(* IEC 61131-3 sources: RL_MAR/experiments/comparison/llm4plc/results/Qwen-Qwen3.5-9B_20260506_150728/20260506_170933, 3 files *)

(* ---- generated_code_iteration_0.st ---- *)
START_ST
FUNCTION_BLOCK BakeryOvenControl
VAR_INPUT
    TemperatureSensor : REAL; (* Sensor input for oven temperature *)
    HumiditySensor : REAL; (* Sensor input for oven humidity *)
    StartSignal : BOOL; (* Input to start the baking process *)
END_VAR
VAR_OUTPUT
    HeatingElement : BOOL; (* Control signal for heating element *)
    CoolingElement : BOOL; (* Control signal for cooling element *)
    HumidityControl : BOOL; (* Control signal for humidity system *)
    DehumidityControl : BOOL; (* Control signal for dehumidification *)
END_VAR
VAR
    OvenTemperature : REAL := 0.0; (* Current oven temperature setpoint *)
    OvenHumidity : REAL := 0.0; (* Current humidity setpoint *)
    BakingTime : TIME := T#0s; (* Total baking time setpoint *)
    OvenStatus : BOOL := FALSE; (* Oven status: TRUE=On, FALSE=Off *)
    HeatingThreshold : REAL := 2.0; (* Temperature control threshold *)
    HumidityThreshold : REAL := 5.0; (* Humidity control threshold *)

    CurrentTemperature : REAL; (* To store the latest sensor reading *)
    CurrentHumidity : REAL; (* To store the latest sensor reading *)
    TimerAccumulator : TIME := T#0s; (* To accumulate time for the 1-second decrement logic *)
    TimerFlag : BOOL := FALSE; (* Flag to indicate if 1 second has elapsed *)
    BakingTimeRemaining : TIME := T#0s; (* Working copy of the baking time to decrement *)

    OneSecondTimer : TON; (* Timer to generate 1-second pulses *)
END_VAR

(* --- State Machine Logic --- *)
CASE OvenStatus OF
    0: (* STATE 0: OFF *)
        (* Initialize/Reset logic *)
        OvenStatus := FALSE;
        BakingTimeRemaining := T#0s;
        TimerAccumulator := T#0s;
        TimerFlag := FALSE;

        (* Ensure all outputs are deactivated *)
        HeatingElement := FALSE;
        CoolingElement := FALSE;
        HumidityControl := FALSE;
        DehumidityControl := FALSE;

        (* Wait for StartSignal to transition to BAKING state *)
        IF StartSignal THEN
            OvenStatus := 1;
        END_IF;

    1: (* STATE 1: BAKING *)
        (* Read Sensor Inputs *)
        CurrentTemperature := TemperatureSensor;
        CurrentHumidity := HumiditySensor;

        (* Temperature Control Logic *)
        (* Activate heating when temp falls below setpoint minus threshold *)
        IF CurrentTemperature < (OvenTemperature - HeatingThreshold) THEN
            HeatingElement := TRUE;
        ELSE
            HeatingElement := FALSE;
        END_IF;

        (* Activate cooling when temp exceeds setpoint plus threshold *)
        IF CurrentTemperature > (OvenTemperature + HeatingThreshold) THEN
            CoolingElement := TRUE;
        ELSE
            CoolingElement := FALSE;
        END_IF;

        (* Humidity Control Logic *)
        (* Activate humidification when humidity falls below setpoint minus threshold *)
        IF CurrentHumidity < (OvenHumidity - HumidityThreshold) THEN
            HumidityControl := TRUE;
        ELSE
            HumidityControl := FALSE;
        END_IF;

        (* Activate dehumidification when humidity exceeds setpoint plus threshold *)
        IF CurrentHumidity > (OvenHumidity + HumidityThreshold) THEN
            DehumidityControl := TRUE;
        ELSE
            DehumidityControl := FALSE;
        END_IF;

        (* Timer Logic for Baking Time *)
        (* Reset accumulator if it has expired or if we just finished a second *)
        IF TimerAccumulator >= T#1s THEN
            TimerAccumulator := T#0s;
            TimerFlag := TRUE;
        END_IF;

        (* Decrement baking time if 1 second has elapsed *)
        IF TimerFlag THEN
            BakingTimeRemaining := BakingTimeRemaining - T#1s;
            TimerFlag := FALSE;
        END_IF;

        (* Check for Baking Complete *)
        IF BakingTimeRemaining <= T#0s THEN
            OvenStatus := 0; (* Transition back to OFF state *)
            HeatingElement := FALSE;
            CoolingElement := FALSE;
            HumidityControl := FALSE;
            DehumidityControl := FALSE;
        END_IF;
END_CASE

(* --- Internal Timer Logic for 1-second Pulse --- *)
(* This timer generates a pulse every second to drive the decrement logic *)
OneSecondTimer(IN := TimerFlag, PT := T#1s);
(* Note: In this specific logic flow, TimerFlag acts as the trigger.
   A standard TON with IN set to TRUE every scan would work,
   but the accumulator approach above handles the 1s interval cleanly.
   If strict edge-triggering is needed, OneSecondTimer(IN := TRUE, PT:=T#1s)
   would set a done bit, but the accumulator logic above is robust for time-based decrement. *)

END_FUNCTION_BLOCK
END_ST

(* ---- generated_code_iteration_1.st ---- *)
START_REASON
The error "不能将类型 'BOOL' 转换为类型'ANY_INT'" (Cannot convert type 'BOOL' to type 'ANY_INT') occurs in the `CASE OvenStatus OF` statement. In Structured Text (ST), `CASE` statements require the selector expression to be of an integer type (e.g., `INT`, `DINT`, `ANY_INT`) or an enumerated type. The variable `OvenStatus` is declared as `BOOL`. While `FALSE` and `TRUE` are valid, they are not directly compatible with the integer-based selector logic of a `CASE` statement in strict compilers like CODESYS without explicit casting or changing the variable type.

To fix this while maintaining the `FUNCTION_BLOCK` structure and avoiding type casting issues, I will change the internal state representation from `BOOL` to `INT` (using 0 for OFF and 1 for BAKING). This aligns perfectly with the `CASE` statement requirements and resolves the type mismatch error. I will also ensure all variable declarations use `END_VAR` correctly and remove any invalid syntax.
END_REASON

START_ST
FUNCTION_BLOCK BakeryOvenControl
VAR_INPUT
    TemperatureSensor : REAL; (* Sensor input for oven temperature *)
    HumiditySensor : REAL; (* Sensor input for oven humidity *)
    StartSignal : BOOL; (* Input to start the baking process *)
END_VAR
VAR_OUTPUT
    HeatingElement : BOOL; (* Control signal for heating element *)
    CoolingElement : BOOL; (* Control signal for cooling element *)
    HumidityControl : BOOL; (* Control signal for humidity system *)
    DehumidityControl : BOOL; (* Control signal for dehumidification *)
END_VAR
VAR
    OvenStatus : INT := 0; (* Current oven status: 0=OFF, 1=On, 2=Error *)
    OvenTemperature : REAL := 0.0; (* Current oven temperature setpoint *)
    OvenHumidity : REAL := 0.0; (* Current humidity setpoint *)
    BakingTime : TIME := T#0s; (* Total baking time setpoint *)

    CurrentTemperature : REAL; (* To store the latest sensor reading *)
    CurrentHumidity : REAL; (* To store the latest sensor reading *)
    TimerAccumulator : TIME := T#0s; (* To accumulate time for the 1-second decrement logic *)
    TimerFlag : BOOL := FALSE; (* Flag to indicate if 1 second has elapsed *)
    BakingTimeRemaining : TIME := T#0s; (* Working copy of the baking time to decrement *)

    OneSecondTimer : TON; (* Timer to generate 1-second pulses *)
END_VAR

(* --- State Machine Logic --- *)
CASE OvenStatus OF
    0: (* STATE 0: OFF *)
        (* Initialize/Reset logic *)
        OvenStatus := 0;
        BakingTimeRemaining := T#0s;
        TimerAccumulator := T#0s;
        TimerFlag := FALSE;

        (* Ensure all outputs are deactivated *)
        HeatingElement := FALSE;
        CoolingElement := FALSE;
        HumidityControl := FALSE;
        DehumidityControl := FALSE;

        (* Wait for StartSignal to transition to BAKING state *)
        IF StartSignal THEN
            OvenStatus := 1;
        END_IF;

    1: (* STATE 1: BAKING *)
        (* Read Sensor Inputs *)
        CurrentTemperature := TemperatureSensor;
        CurrentHumidity := HumiditySensor;

        (* Temperature Control Logic *)
        (* Activate heating when temp falls below setpoint minus threshold *)
        IF CurrentTemperature < (OvenTemperature - HeatingThreshold) THEN
            HeatingElement := TRUE;
        ELSE
            HeatingElement := FALSE;
        END_IF;

        (* Activate cooling when temp exceeds setpoint plus threshold *)
        IF CurrentTemperature > (OvenTemperature + HeatingThreshold) THEN
            CoolingElement := TRUE;
        ELSE
            CoolingElement := FALSE;
        END_IF;

        (* Humidity Control Logic *)
        (* Activate humidification when humidity falls below setpoint minus threshold *)
        IF CurrentHumidity < (OvenHumidity - HumidityThreshold) THEN
            HumidityControl := TRUE;
        ELSE
            HumidityControl := FALSE;
        END_IF;

        (* Activate dehumidification when humidity exceeds setpoint plus threshold *)
        IF CurrentHumidity > (OvenHumidity + HumidityThreshold) THEN
            DehumidityControl := TRUE;
        ELSE
            DehumidityControl := FALSE;
        END_IF;

        (* Timer Logic for Baking Time *)
        (* Reset accumulator if it has expired or if we just finished a second *)
        IF TimerAccumulator >= T#1s THEN
            TimerAccumulator := T#0s;
            TimerFlag := TRUE;
        END_IF;

        (* Decrement baking time if 1 second has elapsed *)
        IF TimerFlag THEN
            BakingTimeRemaining := BakingTimeRemaining - T#1s;
            TimerFlag := FALSE;
        END_IF;

        (* Check for Baking Complete *)
        IF BakingTimeRemaining <= T#0s THEN
            OvenStatus := 0; (* Transition back to OFF state *)
            HeatingElement := FALSE;
            CoolingElement := FALSE;
            HumidityControl := FALSE;
            DehumidityControl := FALSE;
        END_IF;
END_CASE

(* --- Internal Timer Logic for 1-second Pulse --- *)
(* This timer generates a pulse every second to drive the decrement logic *)
OneSecondTimer(IN := TRUE, PT := T#1s);

END_FUNCTION_BLOCK
END_ST

(* ---- generated_code_iteration_2.st ---- *)
START_REASON
The previous code failed due to encoding issues (specifically 'gbk' codec errors) caused by the inclusion of Chinese comments like `(* Sensor input for oven temperature *)`. While the logic was sound, the compiler could not parse the file due to these non-ASCII characters in the specified encoding context.

To fix this:
1.  **Remove all Chinese comments**: Replace them with English comments to ensure universal compatibility.
2.  **Verify Variable Declarations**: Ensure all `VAR` sections end with `END_VAR` and no `END_VAR_OUTPUT` or `END_VAR_INPUT` are used.
3.  **Maintain Structure**: Keep the `FUNCTION_BLOCK` structure and the `CASE` statement logic which now correctly uses `INT` for `OvenStatus`.
4.  **Fix Logic**: The previous logic for the timer was slightly redundant (checking `TimerAccumulator` inside the state machine while also calling the TON block). I will streamline the logic to rely primarily on the `TON` timer's `Q` output for the 1-second pulse, which is more efficient and standard in PLC programming.
5.  **Add Missing Thresholds**: The previous code referenced `HeatingThreshold`, `HumidityThreshold`, etc., but did not declare them. I will add these as internal variables.
END_REASON

START_ST
FUNCTION_BLOCK BakeryOvenControl
VAR_INPUT
    TemperatureSensor : REAL;
    HumiditySensor : REAL;
    StartSignal : BOOL;
END_VAR
VAR_OUTPUT
    HeatingElement : BOOL;
    CoolingElement : BOOL;
    HumidityControl : BOOL;
    DehumidityControl : BOOL;
END_VAR
VAR
    OvenStatus : INT := 0; (* 0=OFF, 1=BAKING, 2=ERROR *)
    OvenTemperature : REAL := 200.0; (* Default setpoint *)
    OvenHumidity : REAL := 50.0; (* Default setpoint *)
    BakingTime : TIME := T#30m;

    CurrentTemperature : REAL;
    CurrentHumidity : REAL;
    TimerAccumulator : TIME := T#0s;
    TimerFlag : BOOL := FALSE;
    BakingTimeRemaining : TIME := T#0s;

    OneSecondTimer : TON;

    (* Thresholds for control logic *)
    HeatingThreshold : REAL := 2.0;
    CoolingThreshold : REAL := 2.0;
    HumidityThreshold : REAL := 5.0;
    DehumidityThreshold : REAL := 5.0;
END_VAR

(* --- State Machine Logic --- *)
CASE OvenStatus OF
    0: (* STATE 0: OFF *)
        OvenStatus := 0;
        BakingTimeRemaining := T#0s;
        TimerAccumulator := T#0s;
        TimerFlag := FALSE;

        (* Ensure all outputs are deactivated *)
        HeatingElement := FALSE;
        CoolingElement := FALSE;
        HumidityControl := FALSE;
        DehumidityControl := FALSE;

        (* Wait for StartSignal to transition to BAKING state *)
        IF StartSignal THEN
            OvenStatus := 1;
        END_IF;

    1: (* STATE 1: BAKING *)
        (* Read Sensor Inputs *)
        CurrentTemperature := TemperatureSensor;
        CurrentHumidity := HumiditySensor;

        (* Temperature Control Logic *)
        IF CurrentTemperature < (OvenTemperature - HeatingThreshold) THEN
            HeatingElement := TRUE;
        ELSE
            HeatingElement := FALSE;
        END_IF;

        IF CurrentTemperature > (OvenTemperature + CoolingThreshold) THEN
            CoolingElement := TRUE;
        ELSE
            CoolingElement := FALSE;
        END_IF;

        (* Humidity Control Logic *)
        IF CurrentHumidity < (OvenHumidity - HumidityThreshold) THEN
            HumidityControl := TRUE;
        ELSE
            HumidityControl := FALSE;
        END_IF;

        IF CurrentHumidity > (OvenHumidity + DehumidityThreshold) THEN
            DehumidityControl := TRUE;
        ELSE
            DehumidityControl := FALSE;
        END_IF;

        (* Timer Logic for Baking Time *)
        (* Use the TON timer output to trigger the 1-second decrement *)
        IF OneSecondTimer.Q THEN
            BakingTimeRemaining := BakingTimeRemaining - T#1s;
            TimerFlag := FALSE;
        END_IF;

        (* Check for Baking Complete *)
        IF BakingTimeRemaining <= T#0s THEN
            OvenStatus := 0; (* Transition back to OFF state *)
            HeatingElement := FALSE;
            CoolingElement := FALSE;
            HumidityControl := FALSE;
            DehumidityControl := FALSE;
        END_IF;
END_CASE

(* --- Internal Timer Logic --- *)
(* This timer generates a pulse every second to drive the decrement logic *)
OneSecondTimer(IN := TRUE, PT := T#1s);

END_FUNCTION_BLOCK
END_ST
